FUNCTION UpdateEventTimestampWithSystemTime
VAR_INPUT
	stEvent : REFERENCE TO ST_Event;
END_VAR
VAR
	fbGETSYSTEMTIME : GETSYSTEMTIME;
	stFileTime : T_FILETIME; // requires Tc2_Utilities
END_VAR

// The function block writes on stFileTime (VAR_OUTPUT) in T_FILETIME format 
fbGETSYSTEMTIME(timeLoDW => stFileTime.dwLowDateTime,
				timeHiDW => stFileTime.dwHighDateTime);

// Overwrites the Timestamp of stEvent using the FILETIME_TO_DT function
stEvent.dtTimestamp := FILETIME_TO_DT(fileTime := stFileTime);

END_FUNCTION

(* stored: Version 1.1.0.1, ProductVersion 3.1.4024.10
   POU UpdateEventTimestampWithSystemTime: Id {de109766-8e59-4882-8690-fd8c87d01dbb}, SpecialFunc None *)
